FUNCTION_BLOCK HandlingSequenceStop EXTENDS HandlingSequence IMPLEMENTS ZCore.ISequence
VAR
  _step : ZCore.Step(HandlingStep.StopBegin, HandlingStep.StopEnd);
  _timerSim : ZAux.Timer;
END_VAR

IF OnStart(_step) THEN
  ; // init custom sequence variables here ...
END_IF

REPEAT
  LogStep();

  CASE _step.Index OF
    (* -------------------------------------------------------------------------------------------------------------------------------- *)
    HandlingStep.StopBegin:
    (* -------------------------------------------------------------------------------------------------------------------------------- *)
      IF _step.OnEntry()
      THEN
        _timerSim.WaitAsync(5);
			END_IF
      
      Await(_timerSim, nextStep:=HandlingStep.StopEnd);
      // _step.SetNext(index:=HandlingStep.StopEnd);

    (* -------------------------------------------------------------------------------------------------------------------------------- *)
    HandlingStep.StopEnd:
    (* -------------------------------------------------------------------------------------------------------------------------------- *)    
      SetBusy(FALSE);
  
  ELSE
    Abort('sequence contains unhandled step');
  END_CASE
UNTIL _step.IsNotRepeatable() OR_ELSE NOT Busy END_REPEAT

END_FUNCTION_BLOCK

(* stored: Version 1.1.0.1
   POU HandlingSequenceStop: Id {f51e7750-1e3b-47bb-bd2e-debde2ea9569}, SpecialFunc None *)
